(* CoDeSys 2.3 export: INFOTASK_PCORCX_VISU.EXP *)
(* Libraries: STANDARD.LIB 5.6.98 11:03:02, TcBase.lib 14.5.09 11:14:08, TcSystem.lib 27.2.12 14:08:36 *)

(* POU InfoTask/P_InfoTask, FBD *)
(****************************************************************************************************************)
(*						Beckhoff Automation Poland								*)
(*								P_InfoTask  v 1.0									*)
(*								22.01.2015										*)
(*_______________________________________________________________________________*)
PROGRAM P_InfoTask
VAR
	arrInfoTask	: ARRAY [1..4] OF FB_InfoTask;
	arrReset		: ARRAY [1..4] OF BOOL;
END_VAR
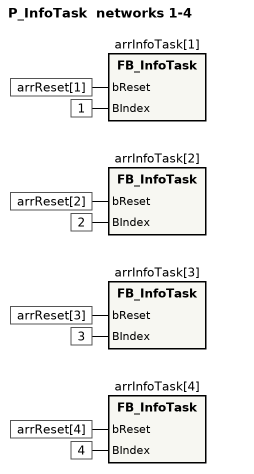
_FBD_ (* Function Block Diagram *)
NETWORK 1
	arrInfoTask[1]:FB_InfoTask(bReset: arrReset[1], BIndex: 1)
NETWORK 2
	arrInfoTask[2]:FB_InfoTask(bReset: arrReset[2], BIndex: 2)
NETWORK 3
	arrInfoTask[3]:FB_InfoTask(bReset: arrReset[3], BIndex: 3)
NETWORK 4
	arrInfoTask[4]:FB_InfoTask(bReset: arrReset[4], BIndex: 4)
_END_FBD_
(* the same logic as Structured Text *)
(* Network 1 *)
arrInfoTask[1](bReset := arrReset[1], BIndex := 1);
(* Network 2 *)
arrInfoTask[2](bReset := arrReset[2], BIndex := 2);
(* Network 3 *)
arrInfoTask[3](bReset := arrReset[3], BIndex := 3);
(* Network 4 *)
arrInfoTask[4](bReset := arrReset[4], BIndex := 4);
END_PROGRAM

(* POU InfoTask/FB_InfoTask, ST *)
(****************************************************************************************************************)
(*						Beckhoff Automation Poland								*)
(*								FB_InfoTask  v 1.0									*)
(*								20.01.2015										*)
(*		Blok funkcyjny FB_InfoTask monitoruje najważniejsze parametry Tasku		 	*)
(*		Zmienna udiCountExceedCycle zlicza liczbę przekroczonych cykli 					*)
(*		zmienna rMaxExceedTime przechowuje maksymalny czas wykonania Tasku		*)
(*		zmienna rAverageCycleTime przechowuje sredni czas wykonania Tasku			*)
(*_______________________________________________________________________________*)
FUNCTION_BLOCK FB_InfoTask
VAR_INPUT
	bReset					: BOOL;						(* Zerowanie zmiennych Persistent*)
	BIndex					: BYTE; 						(* Nr Tasku *)
END_VAR
VAR
	rCycleTime				: REAL;						(* Ustawiony czas Tasku w ms*)
	rLastExecTime			: REAL;						(* Ostatni czas wykonania Tasku w ms*)
	bActive					: BOOL;						 (*Aktywnosc tasku*)
	BPriority					: BYTE;						(*Priorytet tasku*)
	sTaskName				: STRING;					(*Nazwa tasku*)
	bCycleTimeExceeded		: BOOL;						 (*Przekroczenie czasu nastawionego w konfiguracji*)
	rTotalTime				: REAL; 						(*Calkowity czas trwania Tasku *)
	rAverageCycleTime		: REAL;						(* Sredni czas trwania Tasku*)
	rCycleCount				: UDINT; 						(* Calkowita ilosc cykli *)
END_VAR
VAR PERSISTENT
	udiCountExceedCycle		: UDINT; 						(* Licznik przekroczonych cykli *)
	rMaxExecTime			: REAL;						(* Maks czas wykonania Tasku w ms*)
END_VAR
BIndex := LIMIT(1,BIndex,4);
bActive := SystemTaskInfoArr[BIndex].active;

IF bActive THEN
	rCycleTime 		:= UDINT_TO_REAL(SystemTaskInfoArr[BIndex].cycleTime)/10000.0;
	rLastExecTime 	:= UDINT_TO_REAL(SystemTaskInfoArr[BIndex].lastExecTime)/10000.0;
	IF rLastExecTime > rMaxExecTime THEN rMaxExecTime := rLastExecTime; END_IF
	IF SystemTaskInfoArr[BIndex].cycleTimeExceeded  THEN udiCountExceedCycle := udiCountExceedCycle + 1; END_IF
	
	BPriority := SystemTaskInfoArr[BIndex].priority;
	sTaskName := SystemTaskInfoArr[BIndex].taskName;
	bCycleTimeExceeded := SystemTaskInfoArr[BIndex].cycleTimeExceeded;
	
	rCycleCount := rCycleCount + 1;
	rTotalTime := rLastExecTime + rTotalTime;
	rAverageCycleTime := rTotalTime / rCycleCount;
END_IF

IF bReset THEN
	udiCountExceedCycle := 0;
	rMaxExecTime := 0;
	rTotalTime := 0;
	rCycleCount := 0;
	rAverageCycleTime := 0;
	bReset := FALSE;
END_IF
END_FUNCTION_BLOCK

(* Visualisation MAIN_TASKINFO
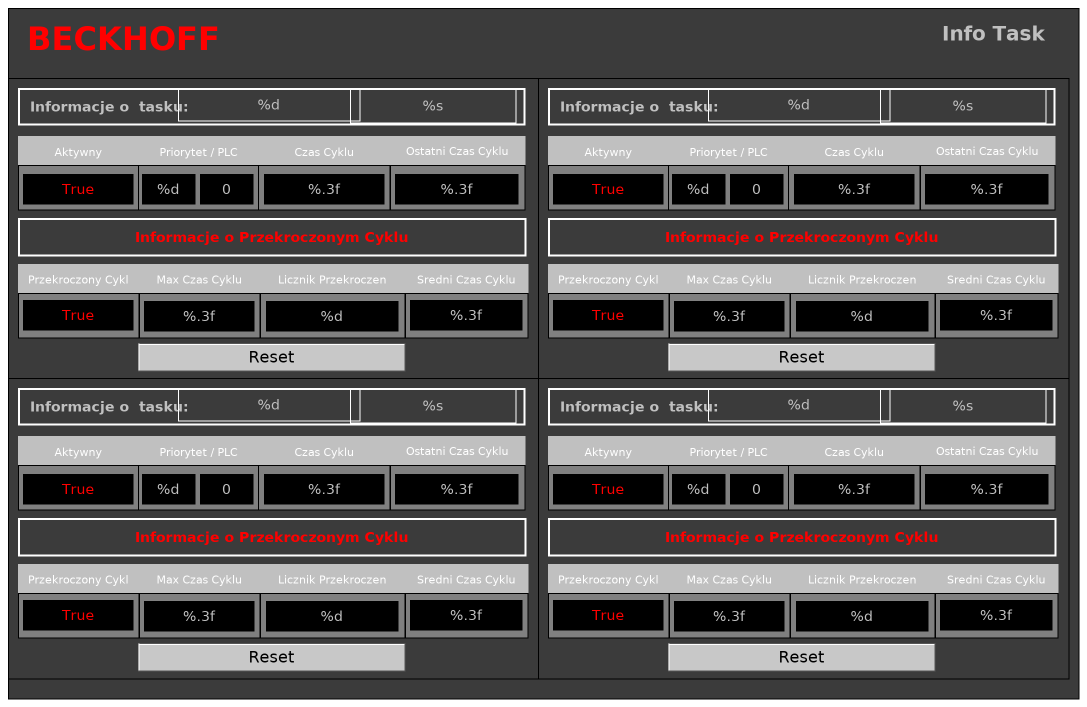
embedded screen at (0,70)-(531,371): PH_TASKINFO
embedded screen at (530,70)-(1061,371): PH_TASKINFO
embedded screen at (0,370)-(531,671): PH_TASKINFO
embedded screen at (530,370)-(1061,671): PH_TASKINFO
rectangle at (910,10)-(1061,41): text "Info Task"
rectangle at (10,10)-(221,51): text "BECKHOFF"
1 more shapes without text or variables
*)

(* Visualisation PH_TASKINFO
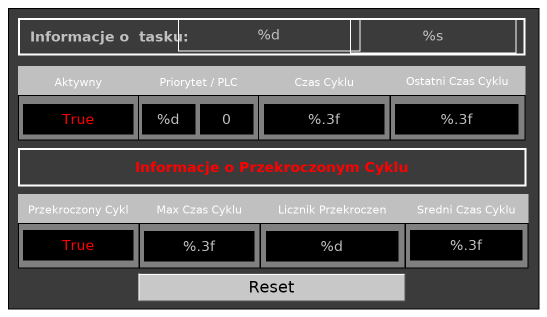
rectangle at (10,10)-(517,47): text "Informacje o  tasku:"
rectangle at (10,140)-(518,178): text "Informacje o Przekroczonym Cyklu"
rectangle at (170,10)-(352,43): text "%d"; shows P_InfoTask.arrInfoTask[$BIndex$].BIndex
rectangle at (342,10)-(508,45): text "%s"; shows P_InfoTask.arrInfoTask[$BIndex$].sTaskName
button at (130,265)-(397,293): text "Reset"; taps P_InfoTask.arrReset[$BIndex$]
rounded rectangle at (10,58)-(131,91): text "Aktywny"
rectangle at (15,96)-(125,126): text "False"; invisible if P_InfoTask.arrInfoTask[$BIndex$].bActive
rectangle at (15,96)-(125,126): text "True"; invisible if NOT P_InfoTask.arrInfoTask[$BIndex$].bActive
rounded rectangle at (130,58)-(251,91): text "Priorytet / PLC"
rectangle at (134,96)-(187,126): text "%d"; shows P_InfoTask.arrInfoTask[$BIndex$].BPriority
rounded rectangle at (250,58)-(383,91): text "Czas Cyklu"
rectangle at (256,96)-(376,126): text "%.3f"; shows P_InfoTask.arrInfoTask[$BIndex$].rCycleTime
rounded rectangle at (382,58)-(517,89): text "Ostatni Czas Cyklu"
rectangle at (387,96)-(510,126): text "%.3f"; shows P_InfoTask.arrInfoTask[$BIndex$].rLastExecTime
rounded rectangle at (10,186)-(131,218): text "Przekroczony Cykl"
rectangle at (15,222)-(125,252): text "False"; invisible if P_InfoTask.arrInfoTask[$BIndex$].bCycleTimeExceeded
rectangle at (15,222)-(125,252): text "True"; invisible if NOT P_InfoTask.arrInfoTask[$BIndex$].bCycleTimeExceeded
rounded rectangle at (131,186)-(252,218): text "Max Czas Cyklu"
rectangle at (136,223)-(246,253): text "%.3f"; shows P_InfoTask.arrInfoTask[$BIndex$].rMaxExecTime
rounded rectangle at (252,186)-(397,218): text "Licznik Przekroczen"
rectangle at (258,223)-(390,253): text "%d"; shows P_InfoTask.arrInfoTask[$BIndex$].udiCountExceedCycle
rounded rectangle at (397,186)-(520,218): text "Sredni Czas Cyklu"
rectangle at (402,222)-(514,252): text "%.3f"; shows P_InfoTask.arrInfoTask[$BIndex$].rAverageCycleTime
rectangle at (192,96)-(245,126): text "%d"; shows P_InfoTask.arrInfoTask[$BIndex$].BPriority - 25; invisible if NOT P_InfoTask.arrInfoTask[$BIndex$].bActive
rectangle at (192,96)-(245,126): text "0"; invisible if P_InfoTask.arrInfoTask[$BIndex$].bActive
9 more shapes without text or variables
*)
